PROGRAM MAIN
VAR
	contador1 : INT;
	contador2 : INT;
	
	contador3 : INT;
END_VAR

contador1 := contador1 + 1;

contador2 := contador2 + 1;
contador2 := contador2 + 1;

contador3 := contador3 + 1;

END_PROGRAM

(* stored: Version 1.1.0.1, ProductVersion 3.1.4024.12
   POU MAIN: Id {46e1726c-ab77-4544-83e9-8f705e970a4a}, SpecialFunc None *)
